// SIMATIC STEP 7 (V5.x) project T13 E29
// CPU: CPU313 C-2 DP(1)
// station: P_ADR_BUS
// station: Hardware
// station: Equipo SIMATIC 300
// program: Programa S7(1)

SYMBOL_TABLE
"AUXILIARES"	DB 1	DB 1
"MARCHA"	I 0.0	BOOL
"FC1"	I 0.1	BOOL
"FC 2"	I 0.2	BOOL
"PARO"	I 0.3	BOOL
"Cycle Execution"	OB 1	OB 1
"CINTA 1"	Q 0.0	BOOL
"LED CINTA 1"	Q 0.1	BOOL
"CINTA 2"	Q 0.2	BOOL
"LED CINTA 2"	Q 0.3	BOOL
"LED PARO"	Q 0.4	BOOL
END_SYMBOL_TABLE

DATA_BLOCK "AUXILIARES"	// DB 1
VERSION : 0.1
  STRUCT
   F0 : BOOL ;
   F1 : BOOL ;
   F2 : BOOL ;
   F3 : BOOL ;
   F4 : BOOL ;
   B5 : BOOL ;
   B6 : BOOL ;
   B7 : BOOL ;
   F10 : BOOL ;
  END_STRUCT ;	
BEGIN
END_DATA_BLOCK

ORGANIZATION_BLOCK "Cycle Execution"	// OB 1
TITLE = "Main Program Sweep (Cycle)"
//MANUFACTURA.
VERSION : 0.1
VAR_TEMP
  OB1_EV_CLASS : BYTE ;	//Bits 0-3 = 1 (Coming event), Bits 4-7 = 1 (Event class 1)
  OB1_SCAN_1 : BYTE ;	//1 (Cold restart scan 1 of OB 1), 3 (Scan 2-n of OB 1)
  OB1_PRIORITY : BYTE ;	//Priority of OB Execution
  OB1_OB_NUMBR : BYTE ;	//1 (Organization block 1, OB1)
  OB1_RESERVED_1 : BYTE ;	//Reserved for system
  OB1_RESERVED_2 : BYTE ;	//Reserved for system
  OB1_PREV_CYCLE : INT ;	//Cycle time of previous OB1 scan (milliseconds)
  OB1_MIN_CYCLE : INT ;	//Minimum cycle time of OB1 (milliseconds)
  OB1_MAX_CYCLE : INT ;	//Maximum cycle time of OB1 (milliseconds)
  OB1_DATE_TIME : DATE_AND_TIME ;	//Date and time OB1 started
END_VAR
BEGIN
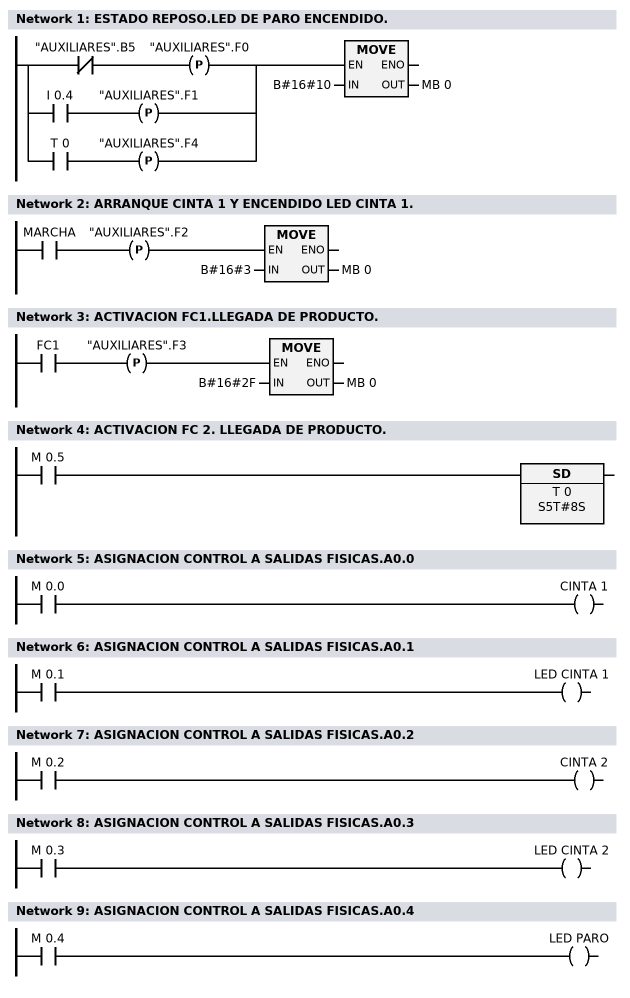
NETWORK
TITLE = ESTADO REPOSO.LED DE PARO ENCENDIDO.
      A(;
      AN    "AUXILIARES".B5;
      FP    "AUXILIARES".F0;
      O(;
      A     I 0.4;
      FP    "AUXILIARES".F1;
      );
      O(;
      A     T 0;
      FP    "AUXILIARES".F4;
      );
      );
      JNB   _001;
      L     B#16#10;
      T     MB 0;
_001: NOP   0;
NETWORK
TITLE = ARRANQUE CINTA 1 Y ENCENDIDO LED CINTA 1.
      A     "MARCHA";
      FP    "AUXILIARES".F2;
      JNB   _002;
      L     B#16#3;
      T     MB 0;
_002: NOP   0;
NETWORK
TITLE = ACTIVACION FC1.LLEGADA DE PRODUCTO.
//SE ACTIVARAN CINTA 2 Y LED CINTA 2.
      A     "FC1";
      FP    "AUXILIARES".F3;
      JNB   _003;
      L     B#16#2F;
      T     MB 0;
_003: NOP   0;
NETWORK
TITLE = ACTIVACION FC 2. LLEGADA DE PRODUCTO.
//EMPIEZA ACONTAR UN TIEMPO DE DESCONEXION QUE SERA DE 8S.UTILIZO M0.5 PARA 
//ALIMENTAR EL TEMPORIZADOR.
      A     M 0.5;
      L     S5T#8S;
      SD    T 0;
NETWORK
TITLE = ASIGNACION CONTROL A SALIDAS FISICAS.A0.0
      A     M 0.0;
      =     "CINTA 1";
NETWORK
TITLE = ASIGNACION CONTROL A SALIDAS FISICAS.A0.1
      A     M 0.1;
      =     "LED CINTA 1";
NETWORK
TITLE = ASIGNACION CONTROL A SALIDAS FISICAS.A0.2
      A     M 0.2;
      =     "CINTA 2";
NETWORK
TITLE = ASIGNACION CONTROL A SALIDAS FISICAS.A0.3
      A     M 0.3;
      =     "LED CINTA 2";
NETWORK
TITLE = ASIGNACION CONTROL A SALIDAS FISICAS.A0.4
      A     M 0.4;
      =     "LED PARO";
END_ORGANIZATION_BLOCK
